ABB RAPID module: Light Drawing

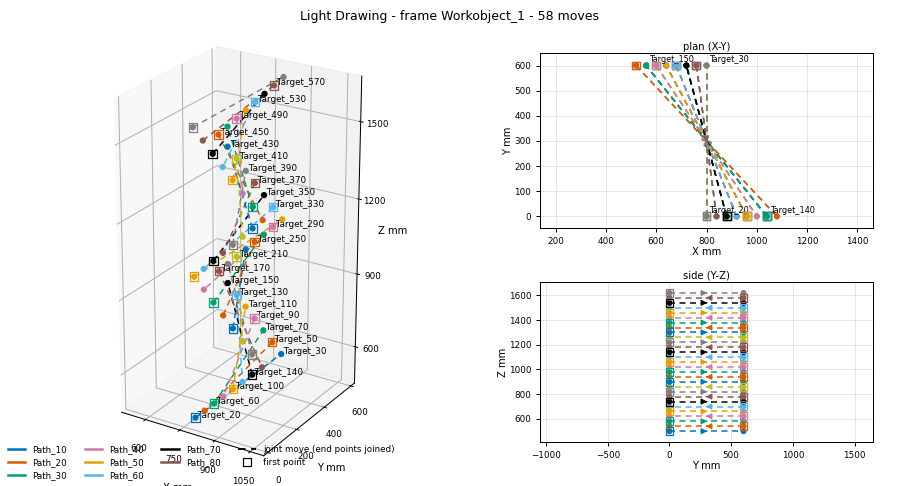
[picture p0: tool path of Light Drawing in frame Workobject_1, 58 of 58 moves have a stored position in this frame; points joined in program order, loops and branches not executed]
# Robotics

MODULE Module1
	CONST robtarget Target_20:=[[800,0,500],[0.49999989,0,0.866025467,0],[0,0,0,0],[9E9,9E9,9E9,9E9,9E9,9E9]];
	CONST robtarget Target_30:=[[800,600,500],[0.49999989,0,0.866025467,0],[0,0,-1,0],[9E9,9E9,9E9,9E9,9E9,9E9]];
	CONST robtarget Target_50:=[[760,600,540],[0.49999989,0,0.866025467,0],[0,0,-1,0],[9E9,9E9,9E9,9E9,9E9,9E9]];
	CONST robtarget Target_40:=[[840,0,540],[0.49999989,0,0.866025467,0],[0,-1,0,0],[9E9,9E9,9E9,9E9,9E9,9E9]];
	CONST robtarget Target_60:=[[880,0,580],[0.49999989,0,0.866025467,0],[0,0,0,0],[9E9,9E9,9E9,9E9,9E9,9E9]];
	CONST robtarget Target_70:=[[720,600,580],[0.49999989,0,0.866025467,0],[0,0,-1,0],[9E9,9E9,9E9,9E9,9E9,9E9]];
	CONST robtarget Target_90:=[[680,600,620],[0.49999989,0,0.866025467,0],[0,0,-1,0],[9E9,9E9,9E9,9E9,9E9,9E9]];
	CONST robtarget Target_80:=[[920,0,620],[0.49999989,0,0.866025467,0],[0,-1,0,0],[9E9,9E9,9E9,9E9,9E9,9E9]];
	CONST robtarget Target_100:=[[960,0,660],[0.49999989,0,0.866025467,0],[0,0,0,0],[9E9,9E9,9E9,9E9,9E9,9E9]];
	CONST robtarget Target_110:=[[640,600,660],[0.49999989,0,0.866025467,0],[0,0,-1,0],[9E9,9E9,9E9,9E9,9E9,9E9]];
	CONST robtarget Target_130:=[[600,600,700],[0.49999989,0,0.866025467,0],[0,0,-1,0],[9E9,9E9,9E9,9E9,9E9,9E9]];
	CONST robtarget Target_120:=[[1000,0,700],[0.49999989,0,0.866025467,0],[0,0,0,0],[9E9,9E9,9E9,9E9,9E9,9E9]];
	CONST robtarget Target_140:=[[1040,0,740],[0.49999989,0,0.866025467,0],[0,0,0,0],[9E9,9E9,9E9,9E9,9E9,9E9]];
	CONST robtarget Target_150:=[[560,600,740],[0.49999989,0,0.866025467,0],[0,0,-1,0],[9E9,9E9,9E9,9E9,9E9,9E9]];
	CONST robtarget Target_170:=[[520,600,780],[0.49999989,0,0.866025467,0],[0,0,-1,0],[9E9,9E9,9E9,9E9,9E9,9E9]];
	CONST robtarget Target_160:=[[1080,0,780],[0.49999989,0,0.866025467,0],[0,-1,0,0],[9E9,9E9,9E9,9E9,9E9,9E9]];
	CONST robtarget Target_180:=[[1040,0,820],[0.49999989,0,0.866025467,0],[0,0,0,0],[9E9,9E9,9E9,9E9,9E9,9E9]];
	CONST robtarget Target_190:=[[560,600,820],[0.49999989,0,0.866025467,0],[0,0,-1,0],[9E9,9E9,9E9,9E9,9E9,9E9]];
	CONST robtarget Target_210:=[[600,600,860],[0.49999989,0,0.866025467,0],[0,0,-1,0],[9E9,9E9,9E9,9E9,9E9,9E9]];
	CONST robtarget Target_200:=[[1000,0,860],[0.49999989,0,0.866025467,0],[0,-1,0,0],[9E9,9E9,9E9,9E9,9E9,9E9]];
	CONST robtarget Target_220:=[[960,0,900],[0.49999989,0,0.866025467,0],[0,0,0,0],[9E9,9E9,9E9,9E9,9E9,9E9]];
	CONST robtarget Target_230:=[[640,600,900],[0.49999989,0,0.866025467,0],[0,1,-1,0],[9E9,9E9,9E9,9E9,9E9,9E9]];
	CONST robtarget Target_250:=[[680,600,940],[0.49999989,0,0.866025467,0],[0,1,-1,0],[9E9,9E9,9E9,9E9,9E9,9E9]];
	CONST robtarget Target_240:=[[920,0,940],[0.49999989,0,0.866025467,0],[0,-1,0,0],[9E9,9E9,9E9,9E9,9E9,9E9]];
	CONST robtarget Target_260:=[[880,0,980],[0.49999989,0,0.866025467,0],[0,0,0,0],[9E9,9E9,9E9,9E9,9E9,9E9]];
	CONST robtarget Target_270:=[[720,600,980],[0.49999989,0,0.866025467,0],[0,1,-1,0],[9E9,9E9,9E9,9E9,9E9,9E9]];
	CONST robtarget Target_290:=[[760,600,1020],[0.49999989,0,0.866025467,0],[0,1,-1,0],[9E9,9E9,9E9,9E9,9E9,9E9]];
	CONST robtarget Target_280:=[[840,0,1020],[0.49999989,0,0.866025467,0],[0,2,-3,0],[9E9,9E9,9E9,9E9,9E9,9E9]];
	CONST robtarget Target_300:=[[800,0,1060],[0.49999989,0,0.866025467,0],[0,-2,-2,0],[9E9,9E9,9E9,9E9,9E9,9E9]];
	CONST robtarget Target_310:=[[800,600,1060],[0.49999989,0,0.866025467,0],[0,1,-1,0],[9E9,9E9,9E9,9E9,9E9,9E9]];
	CONST robtarget Target_330:=[[760,600,1100],[0.49999989,0,0.866025467,0],[0,1,-2,0],[9E9,9E9,9E9,9E9,9E9,9E9]];
	CONST robtarget Target_320:=[[840,0,1100],[0.49999989,0,0.866025467,0],[0,2,-3,0],[9E9,9E9,9E9,9E9,9E9,9E9]];
	CONST robtarget Target_340:=[[880,0,1140],[0.49999989,0,0.866025467,0],[0,-2,-2,0],[9E9,9E9,9E9,9E9,9E9,9E9]];
	CONST robtarget Target_350:=[[720,600,1140],[0.49999989,0,0.866025467,0],[0,1,-2,0],[9E9,9E9,9E9,9E9,9E9,9E9]];
	CONST robtarget Target_370:=[[680,600,1180],[0.49999989,0,0.866025467,0],[0,1,-2,0],[9E9,9E9,9E9,9E9,9E9,9E9]];
	CONST robtarget Target_360:=[[920,0,1180],[0.49999989,0,0.866025467,0],[0,2,-3,0],[9E9,9E9,9E9,9E9,9E9,9E9]];
	CONST robtarget Target_380:=[[960,0,1220],[0.49999989,0,0.866025467,0],[0,-2,-2,0],[9E9,9E9,9E9,9E9,9E9,9E9]];
	CONST robtarget Target_390:=[[640,600,1220],[0.49999989,0,0.866025467,0],[0,1,-2,0],[9E9,9E9,9E9,9E9,9E9,9E9]];
	CONST robtarget Target_410:=[[600,600,1260],[0.49999989,0,0.866025467,0],[0,1,-2,0],[9E9,9E9,9E9,9E9,9E9,9E9]];
	CONST robtarget Target_400:=[[1000,0,1260],[0.49999989,0,0.866025467,0],[0,2,-3,0],[9E9,9E9,9E9,9E9,9E9,9E9]];
	CONST robtarget Target_420:=[[1040,0,1300],[0.49999989,0,0.866025467,0],[0,-2,-2,0],[9E9,9E9,9E9,9E9,9E9,9E9]];
	CONST robtarget Target_430:=[[560,600,1300],[0.49999989,0,0.866025467,0],[0,1,-2,0],[9E9,9E9,9E9,9E9,9E9,9E9]];
	CONST robtarget Target_450:=[[520,600,1340],[0.49999989,0,0.866025467,0],[0,1,-2,0],[9E9,9E9,9E9,9E9,9E9,9E9]];
	CONST robtarget Target_440:=[[1080,0,1340],[0.49999989,0,0.866025467,0],[-1,2,-3,0],[9E9,9E9,9E9,9E9,9E9,9E9]];
	CONST robtarget Target_460:=[[1040,0,1380],[0.49999989,0,0.866025467,0],[0,-2,-2,0],[9E9,9E9,9E9,9E9,9E9,9E9]];
	CONST robtarget Target_470:=[[560,600,1380],[0.49999989,0,0.866025467,0],[0,1,-2,0],[9E9,9E9,9E9,9E9,9E9,9E9]];
	CONST robtarget Target_490:=[[600,600,1420],[0.49999989,0,0.866025467,0],[0,1,-2,0],[9E9,9E9,9E9,9E9,9E9,9E9]];
	CONST robtarget Target_480:=[[1000,0,1420],[0.49999989,0,0.866025467,0],[-1,2,-3,0],[9E9,9E9,9E9,9E9,9E9,9E9]];
	CONST robtarget Target_500:=[[960,0,1460],[0.49999989,0,0.866025467,0],[0,-2,-2,0],[9E9,9E9,9E9,9E9,9E9,9E9]];
	CONST robtarget Target_510:=[[640,600,1460],[0.49999989,0,0.866025467,0],[0,1,-2,0],[9E9,9E9,9E9,9E9,9E9,9E9]];
	CONST robtarget Target_530:=[[680,600,1500],[0.49999989,0,0.866025467,0],[0,1,-2,0],[9E9,9E9,9E9,9E9,9E9,9E9]];
	CONST robtarget Target_520:=[[920,0,1500],[0.49999989,0,0.866025467,0],[-1,2,-3,0],[9E9,9E9,9E9,9E9,9E9,9E9]];
	CONST robtarget Target_540:=[[880,0,1540],[0.49999989,0,0.866025467,0],[0,-2,-2,0],[9E9,9E9,9E9,9E9,9E9,9E9]];
	CONST robtarget Target_550:=[[720,600,1540],[0.49999989,0,0.866025467,0],[0,1,-2,0],[9E9,9E9,9E9,9E9,9E9,9E9]];
	CONST robtarget Target_570:=[[760,600,1580],[0.49999989,0,0.866025467,0],[0,1,-2,0],[9E9,9E9,9E9,9E9,9E9,9E9]];
	CONST robtarget Target_560:=[[840,0,1580],[0.49999989,0,0.866025467,0],[-1,2,-3,0],[9E9,9E9,9E9,9E9,9E9,9E9]];
	CONST robtarget Target_580:=[[800,0,1620],[0.49999989,0,0.866025467,0],[0,-2,-2,0],[9E9,9E9,9E9,9E9,9E9,9E9]];
	CONST robtarget Target_590:=[[800,600,1620],[0.49999989,0,0.866025467,0],[0,1,-2,0],[9E9,9E9,9E9,9E9,9E9,9E9]];
	PROC Path_10()
	    MoveJ Target_20,v1000,z100,tool0\WObj:=Workobject_1;
	    MoveJ Target_30,v1000,z100,tool0\WObj:=Workobject_1;
	ENDPROC
	PROC Path_20()
	    MoveJ Target_50,v1000,z100,tool0\WObj:=Workobject_1;
	    MoveJ Target_40,v1000,z100,tool0\WObj:=Workobject_1;
	ENDPROC
	PROC Path_30()
	    MoveJ Target_60,v1000,z100,tool0\WObj:=Workobject_1;
	    MoveJ Target_70,v1000,z100,tool0\WObj:=Workobject_1;
	ENDPROC
	PROC Path_40()
	    MoveJ Target_90,v1000,z100,tool0\WObj:=Workobject_1;
	    MoveJ Target_80,v1000,z100,tool0\WObj:=Workobject_1;
	ENDPROC
	PROC Path_50()
	    MoveJ Target_100,v1000,z100,tool0\WObj:=Workobject_1;
	    MoveJ Target_110,v1000,z100,tool0\WObj:=Workobject_1;
	ENDPROC
	PROC Path_60()
	    MoveJ Target_130,v1000,z100,tool0\WObj:=Workobject_1;
	    MoveJ Target_120,v1000,z100,tool0\WObj:=Workobject_1;
	ENDPROC
	PROC Path_70()
	    MoveJ Target_140,v1000,z100,tool0\WObj:=Workobject_1;
	    MoveJ Target_150,v1000,z100,tool0\WObj:=Workobject_1;
	ENDPROC
	PROC Path_80()
	    MoveJ Target_170,v1000,z100,tool0\WObj:=Workobject_1;
	    MoveJ Target_160,v1000,z100,tool0\WObj:=Workobject_1;
	ENDPROC
	PROC Path_90()
	    MoveJ Target_180,v1000,z100,tool0\WObj:=Workobject_1;
	    MoveJ Target_190,v1000,z100,tool0\WObj:=Workobject_1;
	ENDPROC
	PROC Path_100()
	    MoveJ Target_210,v1000,z100,tool0\WObj:=Workobject_1;
	    MoveJ Target_200,v1000,z100,tool0\WObj:=Workobject_1;
	ENDPROC
	PROC Path_110()
	    MoveJ Target_220,v1000,z100,tool0\WObj:=Workobject_1;
	    MoveJ Target_230,v1000,z100,tool0\WObj:=Workobject_1;
	ENDPROC
	PROC Path_120()
	    MoveJ Target_250,v1000,z100,tool0\WObj:=Workobject_1;
	    MoveJ Target_240,v1000,z100,tool0\WObj:=Workobject_1;
	ENDPROC
	PROC Path_130()
	    MoveJ Target_260,v1000,z100,tool0\WObj:=Workobject_1;
	    MoveJ Target_270,v1000,z100,tool0\WObj:=Workobject_1;
	ENDPROC
	PROC Path_140()
	    MoveJ Target_290,v1000,z100,tool0\WObj:=Workobject_1;
	    MoveJ Target_280,v1000,z100,tool0\WObj:=Workobject_1;
	ENDPROC
	PROC Path_150()
	    MoveJ Target_300,v1000,z100,tool0\WObj:=Workobject_1;
	    MoveJ Target_310,v1000,z100,tool0\WObj:=Workobject_1;
	ENDPROC
	PROC Path_160()
	    MoveJ Target_330,v1000,z100,tool0\WObj:=Workobject_1;
	    MoveJ Target_320,v1000,z100,tool0\WObj:=Workobject_1;
	ENDPROC
	PROC Path_170()
	    MoveJ Target_340,v1000,z100,tool0\WObj:=Workobject_1;
	    MoveJ Target_350,v1000,z100,tool0\WObj:=Workobject_1;
	ENDPROC
	PROC Path_180()
	    MoveJ Target_370,v1000,z100,tool0\WObj:=Workobject_1;
	    MoveJ Target_360,v1000,z100,tool0\WObj:=Workobject_1;
	ENDPROC
	PROC Path_190()
	    MoveJ Target_380,v1000,z100,tool0\WObj:=Workobject_1;
	    MoveJ Target_390,v1000,z100,tool0\WObj:=Workobject_1;
	ENDPROC
	PROC Path_200()
	    MoveJ Target_410,v1000,z100,tool0\WObj:=Workobject_1;
	    MoveJ Target_400,v1000,z100,tool0\WObj:=Workobject_1;
	ENDPROC
	PROC Path_210()
	    MoveJ Target_420,v1000,z100,tool0\WObj:=Workobject_1;
	    MoveJ Target_430,v1000,z100,tool0\WObj:=Workobject_1;
	ENDPROC
	PROC Path_220()
	    MoveJ Target_450,v1000,z100,tool0\WObj:=Workobject_1;
	    MoveJ Target_440,v1000,z100,tool0\WObj:=Workobject_1;
	ENDPROC
	PROC Path_230()
	    MoveJ Target_460,v1000,z100,tool0\WObj:=Workobject_1;
	    MoveJ Target_470,v1000,z100,tool0\WObj:=Workobject_1;
	ENDPROC
	PROC Path_240()
	    MoveJ Target_490,v1000,z100,tool0\WObj:=Workobject_1;
	    MoveJ Target_480,v1000,z100,tool0\WObj:=Workobject_1;
	ENDPROC
	PROC Path_250()
	    MoveJ Target_500,v1000,z100,tool0\WObj:=Workobject_1;
	    MoveJ Target_510,v1000,z100,tool0\WObj:=Workobject_1;
	ENDPROC
	PROC Path_260()
	    MoveJ Target_530,v1000,z100,tool0\WObj:=Workobject_1;
	    MoveJ Target_520,v1000,z100,tool0\WObj:=Workobject_1;
	ENDPROC
	PROC Path_270()
	    MoveJ Target_540,v1000,z100,tool0\WObj:=Workobject_1;
	    MoveJ Target_550,v1000,z100,tool0\WObj:=Workobject_1;
	ENDPROC
	PROC Path_280()
	    MoveJ Target_570,v1000,z100,tool0\WObj:=Workobject_1;
	    MoveJ Target_560,v1000,z100,tool0\WObj:=Workobject_1;
	ENDPROC
	PROC Path_290()
	    MoveJ Target_580,v1000,z100,tool0\WObj:=Workobject_1;
	    MoveJ Target_590,v1000,z100,tool0\WObj:=Workobject_1;
	ENDPROC
    PROC main()
        Path_10;
        Path_20;
         Path_30;
        Path_40;
        Path_50;
        Path_60;
        Path_70;
        Path_80;
        Path_90;
        Path_100;
        Path_110;
        Path_120;
        Path_130;
        Path_140;
        Path_150;
        Path_160;
        Path_170;
        Path_180;
        Path_190;
        Path_200;
        Path_210;
        Path_220;
        Path_230;
        Path_240;
        Path_250;
        Path_260;
        Path_270;
        Path_280;
        Path_290;

    ENDPROC
ENDMODULE
